Staubli VAL3: NULLKEY.pgx

public program nullKey(num& x_nKey[])
begin
  //-----------------------------------------------------------------------
  //Header begin
  //  Wait a new key was pressed, and put x_nKey to 0.
  //  This program was used for waiting the release of a button.
  //
  //Input parameter
  //  num x_nKey :
  //    role : this variable is put to 0 when a new key was pressed.
  //
  //History
  //  Creation : 28-04-08 - f.Rob
  //Header end
  //-----------------------------------------------------------------------
  //Wait a new key stroke
  wait(getKey()==-1)
  x_nKey=0
end
